Program P30_ManualControl
VAR
	analogDeviceRampControl : FB_AnalogDeviceRampControl;
END_VAR

analogDeviceRampControl();

END_PROGRAM

(* stored: Version 1.1.0.1, ProductVersion 3.1.4024.15
   POU P30_ManualControl: Id {1bb09c77-6d3f-460c-8adf-a95106aac779}, SpecialFunc None *)
